{attribute addProperty BoxType "EL1512-0000-0017"}
{attribute addProperty Id "CNT_Inputs_ChannelAT %I*ARRAY[0..1] OF CNT_Inputs_Channel_D5E647EE96120CNT_Outputs_ChannelAT %Q*ARRAY[0..1] OF CNT_Outputs_Channel_C7399CE196120WcStateAT %I*WcState_F855686C1620InfoDataAT %I*InfoData_BC63D37F80100"}
{attribute addProperty CRC "3919822883"}
{attribute addProperty SizeInBites "288"}
{attribute addProperty SizeInBytes "36"}
TYPE EL1512_C3D5AB70 :
STRUCT
	{attribute addProperty Name "CNT_Inputs_Channel"}
	CNT_Inputs_Channel : ARRAY[0..1] OF CNT_Inputs_Channel_D5E647EE;
	{attribute addProperty Name "CNT_Outputs_Channel"}
	CNT_Outputs_Channel : ARRAY[0..1] OF CNT_Outputs_Channel_C7399CE1;
	{attribute addProperty Name "WcState"}
	WcState : WcState_F855686C;
	{attribute addProperty Name "InfoData"}
	InfoData : InfoData_BC63D37F;
END_STRUCT
END_TYPE

(* stored: Version 1.2.0.0, ProductVersion 3.1.4024.9
   DUT EL1512_C3D5AB70: Id {dc2dfea9-fd3d-4d82-b9f5-441c38e13c81} *)
